Universal Robots PolyScope program: g_to_c.urp

Program g_to_c (installation=string_planes directory=/programs/string_crossings createdIn=5.17.3 lastSavedIn=5.17.3 robotSerialNumber=20245501435)
Calibrated DH parameters: a=[0.000154, -0.137004, -0.385524, -0.00002, 0.000092, 0]; d=[0.162441, 211.794786, -230.585024, 18.923638, 0.099786, 0.09951]; alpha=[1.569493, -0.001902, 0.003874, 1.570111, -1.570167, 0]; deltaTheta=[0, -1.242934, 1.056292, 0.186646, 0.000002, 0.000001]
InitVariablesNode
Robot Program (runOnlyOnce=false)
  bow_section := -1
  If bow_section≟-1
    MoveJ speed 60 deg/s, acceleration 80 deg/s^2 (useActiveTCP=true) feature=Base
      Waypoint Waypoint_2 (Relative): relativeFromPosition TCP in base x=333.313 y=655.493 z=103.664 mm, rx=-1.6491 ry=-1.7981 rz=0.6657 rad; joints [-132.463, -27.758, 71.844, -100.481, -56.042, -147.727] deg; TCP offset x=28.21 y=-96.107 z=-99.69 mm, rx=0 ry=0 rz=0 rad; TCP in base x=245.295 y=570.7 z=53.28 mm, rx=-1.8424 ry=-1.3918 rz=0.0687 rad; joints [-132.227, -24.799, 96.314, -169.321, -42.687, -112.61] deg
  ElseIf bow_section≟0
    MoveJ speed 60 deg/s, acceleration 80 deg/s^2 (useActiveTCP=true) feature=Base
      Waypoint Waypoint_1 (Relative): relativeFromPosition TCP in base x=267.761 y=455.827 z=63.349 mm, rx=-1.6064 ry=-1.9107 rz=0.8701 rad; joints [-141.614, -39.193, 108.912, -115.289, -70.779, -159.12] deg; TCP in base x=195.266 y=411.465 z=21.275 mm, rx=-1.7342 ry=-1.5169 rz=0.4321 rad; joints [-140.231, -30.937, 122.534, -154.989, -45.801, -143.196] deg
  Else 
    MoveJ speed 60 deg/s, acceleration 80 deg/s^2 (useActiveTCP=true) feature=Base
      Waypoint Waypoint_3 (Relative): relativeFromPosition TCP in base x=243.617 y=214.085 z=64.401 mm, rx=-1.5874 ry=-1.9213 rz=0.9621 rad; joints [-169.304, -44.6, 138.123, -133.882, -94.42, -177.774] deg; TCP in base x=152.648 y=275.83 z=-5.999 mm, rx=-1.6122 ry=-1.6008 rz=0.7404 rad; joints [-153.502, -26.651, 138.518, -151.349, -62.642, -165.794] deg
